SUBAPPLICATION Knickdeichsel_Sitzventile (* Subapplication Type *)
  (* Standard: 61499-2 *)
  (* Version 1.0, 2023-02-11, franz *)
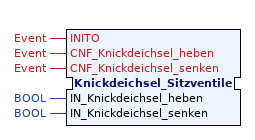
  EVENT_INPUT
    INITO;
    CNF_Knickdeichsel_heben;
    CNF_Knickdeichsel_senken;
  END_EVENT
  VAR_INPUT
    IN_Knickdeichsel_heben : BOOL;
    IN_Knickdeichsel_senken : BOOL;
  END_VAR
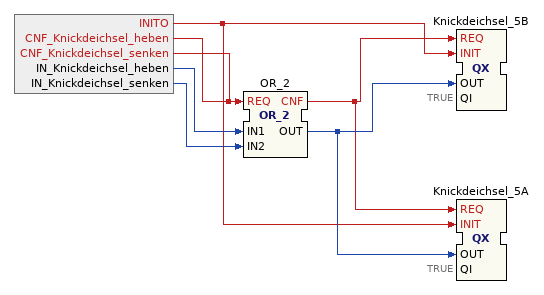
  FBS
    OR_2 : OR_2; {SET_ATTRIBUTE(PinComment, IN1:Knickdeichsel_heben)} {SET_ATTRIBUTE(PinComment, IN2:Knickdeichsel_senken)}
    Knickdeichsel_5B : QX(QI := TRUE);
    Knickdeichsel_5A : QX(QI := TRUE);
  END_FBS
  EVENT_CONNECTIONS
    OR_2.CNF TO Knickdeichsel_5B.REQ;
    OR_2.CNF TO Knickdeichsel_5A.REQ;
    CNF_Knickdeichsel_heben TO OR_2.REQ;
    CNF_Knickdeichsel_senken TO OR_2.REQ;
    INITO TO Knickdeichsel_5B.INIT;
    INITO TO Knickdeichsel_5A.INIT;
  END_CONNECTIONS
  DATA_CONNECTIONS
    OR_2.OUT TO Knickdeichsel_5B.OUT;
    OR_2.OUT TO Knickdeichsel_5A.OUT;
    IN_Knickdeichsel_heben TO OR_2.IN1;
    IN_Knickdeichsel_senken TO OR_2.IN2;
  END_CONNECTIONS
END_SUBAPPLICATION
